TYPE JBOX_Test_Log :
STRUCT
	Index : INT;
	Description : STRING(255);
	Result : STRING(10);
END_STRUCT
END_TYPE

(* stored: Version 1.1.0.1, ProductVersion 3.1.4024.10
   DUT JBOX_Test_Log: Id {3d836bc5-a48d-4607-9825-fefa17475289} *)
